{attribute 'linkalways'} 
{attribute 'no_explicit_call' := 'This FB is a CLASS and must be accessed using methods or properties'}
{attribute 'enable_dynamic_creation'}
FUNCTION_BLOCK Node_F_VN_SubtractImages EXTENDS VisionNode
VAR
    ipSrcImage1 : _ITcVnImage;
    ipSrcImage2 : _ITcVnImage;
    ipDestImage : _ITcVnImage;
    hrPrev : _HRESULT(S_OK);
	hresult : _HRESULT(S_OK);
END_VAR

METHOD PUBLIC  Clone : I_Node
VAR
	pNode : POINTER TO Node_F_VN_SubtractImages;
END_VAR
pNode := __NEW(Node_F_VN_SubtractImages);
Clone := pNode^;
END_METHOD

METHOD FB_init : BOOL
VAR_INPUT
	bInitRetains : BOOL; // if TRUE, the retain variables are initialized (warm start / cold start)
	bInCopyCode : BOOL;  // if TRUE, the instance afterwards gets moved into the copy code (online change)
END_VAR
AddInput('ipSrcImage1', ipSrcImage1);
AddInput('ipSrcImage2', ipSrcImage2);
AddInput('hrPrev', hrPrev);
AddOutput('ipDestImage', ipDestImage);
AddOutput('hresult',hresult);
END_METHOD

METHOD PROTECTED OnExecute : HRESULT
hresult.Value := F_VN_SubtractImages(
    ipSrcImage1 := ipSrcImage1.Value,
    ipSrcImage2 := ipSrcImage2.Value,
	ipDestImage := ipDestImage.Value,
	hrPrev:= hrPrev.Value);
END_METHOD

METHOD PUBLIC PreExecutionCheck
VAR_INPUT
	Check : I_PreExecutionChecks;
END_VAR
IF FAILED(hrPrev.Value) THEN
    RETURN;
END_IF

Check.IsTrue(ipSrcImage1.IsValid, 'ipSrcImage1 must contain an image');
Check.IsTrue(ipSrcImage2.IsValid, 'ipSrcImage2 must contain an image');
END_METHOD

END_FUNCTION_BLOCK

(* stored: Version 1.1.0.1, ProductVersion 3.1.4024.13
   POU Node_F_VN_SubtractImages: Id {3213bbeb-0919-0609-2850-17dc7e204bf0}, SpecialFunc None
   Folder Constructor: Id {b452280f-6a60-02c7-052e-4147f6646ab0}
   Method Clone: Id {936cd559-7ebb-0d4e-2cd7-53e198c33c2e}
   Method FB_init: Id {fbe8c195-015e-0298-24e9-1b2141dfe55a}
   Method OnExecute: Id {50a761e3-1aaa-0a3b-1485-d5d32dcd1f28}
   Method PreExecutionCheck: Id {78d8334f-e146-0ea6-2bd1-8fe88b62e648} *)
